FUNCTION_BLOCK FB_PrgmBasic
VAR_INPUT
	
	EventParameters:	EventParam_Typ;	
	EventHeader:		EventHeader_Typ;	
END_VAR
VAR_OUTPUT
END_VAR
VAR
	LocalEventQ	: Queue;
	LocalEventObj :LocalEvent_Typ;
	GlobalEventObj :LocalEvent_Typ;
	FlagSendEvent :BOOL;
	FlagActive	:BOOL;
	DummyFlowID: DINT := 0;
END_VAR

//Check if Q has elements
IF THIS^.LocalEventQ.EntriesCount >0 AND (FlagSendEvent=FALSE)  THEN
	THIS^.LocalEventQ.Dequeue(ADR(THIS^.GlobalEventObj),SIZEOF(LocalEvent_Typ));
	FlagSendEvent:=TRUE;
END_IF


IF FlagSendEvent THEN
	IF TestAndSet(THIS^.GlobalEventObj.rEvent.Busy) THEN // Check if the event FB is free
		FlagActive:=TRUE;	
	END_IF
	IF FlagActive THEN
//		THIS^.GlobalEventObj.rEvent(pFlowID:=ADR(GlobalEventObj.flowId),pEvPar:=ADR(GlobalEventObj.EventParameters)); //Call the event FB 
		THIS^.GlobalEventObj.rEvent(pEvHeader:=ADR(GlobalEventObj.EventHeader),pEvPar:=ADR(GlobalEventObj.EventParameters)); //Call the event FB 
		IF THIS^.GlobalEventObj.rEvent.Done THEN
			THIS^.GlobalEventObj.rEvent.Done 	:=FALSE;
			THIS^.GlobalEventObj.rEvent.Busy	:=FALSE;//Free FB
			FlagActive:=FALSE;
			FlagSendEvent:=FALSE;
		END_IF
	END_IF
END_IF

METHOD mEventThrow : BOOL
VAR_INPUT
	rEvent : REFERENCE TO EventHelper;
//	pFlowID :POINTER TO DINT;
	pEvHeader: POINTER TO EventHeader_Typ;
	pEvPar: POINTER TO EventParam_Typ;


END_VAR
IF (pEvHeader^.pFlowID = 0) THEN
	pEvHeader^.pFlowID := ADR(DummyFlowID);
END_IF
//Dereference data
LocalEventObj.EventParameters := pEvPar^;
LocalEventObj.rEvent REF= rEvent;
//LocalEventObj.flowId := pFlowID^;
LocalEventObj.EventHeader := pEvHeader^;
	
LocalEventQ.Enqueue(ADR(THIS^.LocalEventObj),SIZEOF(THIS^.LocalEventObj));
mEventThrow:=TRUE;
END_METHOD

END_FUNCTION_BLOCK

(* stored: Version 1.1.0.1, ProductVersion 3.1.4024.3
   POU FB_PrgmBasic: Id {4ef2c2df-db85-090b-3820-276f69240426}, SpecialFunc None
   Method mEventThrow: Id {35a8d1a2-4b72-0540-2950-352ed3318e11} *)
